Universal Robots PolyScope program: start.urp

Program start (installation=20240827 directory=/programs createdIn=5.13.1 lastSavedIn=5.15.1 robotSerialNumber=20245500285)
Calibrated DH parameters: a=[0.000097, -0.210459, -0.026602, 0.000137, 0.000078, 0]; d=[0.162601, 254.180657, -54.076236, -199.970743, 0.099615, 0.099684]; alpha=[1.569796, -0.001455, 0.001957, 1.570525, -1.571561, 0]; deltaTheta=[0, -1.053331, 8.839472, -1.50296, 0.000002, 0]
InitVariablesNode
Robot Program (runOnlyOnce=true)
  SuppressedNode
    Popup Message (haltProgram=false message=please ensure the state inputType=Text)
  Wait Sleep waitTime=0.8
  SuppressedNode
    Halt
  n := 0
  Loop Forever
    Script: n=n+1
    MoveL speed 3000 mm/s, acceleration 6000 mm/s^2 (useActiveTCP=true) feature=Base
      Waypoint 路点_1: TCP in base x=83.4 y=-280.826 z=106.165 mm, rx=-2.2214 ry=-2.2214 rz=0 rad; joints [79.307, -119.168, 139.328, -110.204, -90.008, 79.431] deg; TCP offset x=-0.17 y=0 z=192.95 mm, rx=0 ry=0 rz=0 rad
    If n≥10
      Script: reset=1
      Wait Sleep waitTime=0.2
      Script: reset=0
      Script: n=0
    MoveL speed 60 mm/s, acceleration 600 mm/s^2 (useActiveTCP=true) feature=Base
      Waypoint 路点_3: TCP in base x=83.402 y=-554.591 z=106.172 mm, rx=-2.2215 ry=-2.2215 rz=0.0001 rad; joints [84.678, -77.014, 104.053, -117.084, -90.042, 84.853] deg
        Until EXPRESSION (allowActions=false deceleration=100) ExpressionBranch=tmp[0]>0
    SuppressedNode
      current := get_actual_tcp_pose()
    SuppressedNode
      If current[1]>-0.553 and current[1]<-0.275
        back := pose_add(current, p[0,0.05,0,0,0,0])
        MoveL speed 3000 mm/s, acceleration 6000 mm/s^2 (useActiveTCP=true) feature=Base
          Waypoint Variable (Variable): motionParameters(blendRadius=0.01); variable=back
  MoveL speed 250 mm/s, acceleration 1200 mm/s^2 (useActiveTCP=true) feature=Base
    Waypoint 路点_1: motionParameters(jointSpeed=1.047198 jointAcceleration=1.396263 cartesianSpeed=0.12 cartesianAcceleration=0.8); TCP in base x=83.4 y=-280.826 z=106.165 mm, rx=-2.2214 ry=-2.2214 rz=0 rad; joints [79.307, -119.168, 139.328, -110.204, -90.008, 79.431] deg
Thread Thread_1 (runOnlyOnce=false)
  tmp := p[0,0,0,0,0,0]
  reset := 0
  Loop Forever
    Script file /programs/pose_register.script
      | tmp[0]=read_input_float_register(0)
      | tmp[1]=read_input_float_register(1)
      | tmp[2]=read_input_float_register(2)
      | tmp[3]=read_input_float_register(3)
      | tmp[4]=read_input_float_register(4)
      | tmp[5]=read_input_float_register(5)
    Script: write_output_float_register(0,reset)
    Script: sync()
